TYPE (* A Structure with 1 BYTE *)
  (* Version 1.0, 2024-02-21, Franz Höpfinger, HR Agrartechnik GmbH *)
  PACKAGE logiBUS::utils::conversion::types;
  ST01B : STRUCT
    B_00 : BYTE; (* BYTE 00 *)
  END_STRUCT;
END_TYPE
